(* CoDeSys 2.3 export: KBRD_TIP.EXP *)

(* Data type in Other *)
TYPE kbrd_tip :
(
    off:=0,
    DOWN:=4,
    UP:=8,
    ENTER:=16,
    OUT:=64,
    ALT:=128,
    F1:=1,
    F2:=2,
    F3:=256,
    pusk_stop:=32,
    ALT_F1:=129,
    ALT_F3:=384
);
END_TYPE
